// TwinCAT 3 PLC project Untitled1
// ProgramVersion: 3.1.4024.0
// libraries:
//   Tc2_Standard, * (Beckhoff Automation GmbH)
//   Tc2_System, * (Beckhoff Automation GmbH)
//   Tc3_Module, * (Beckhoff Automation GmbH)
// project tree:
//   Actuator/Actuator/ FB_Actuator.TcPOU (not stored)
//   Actuator/DUTs/ E_ActuatorCommand.TcDUT, ST_Inputs.TcDUT, ST_Outputs.TcDUT, ST_ActuatorStatus.TcDUT (not stored), ST_ActuatorConfiguration.TcDUT (not stored)
//   Actuator/GVLs/ Param_Actuator.TcGVL
//   Actuator/ ITF_Actuator.TcIO (not stored)
//   Error/DUTs/ E_ErrorPriority.TcDUT, ST_Error.TcDUT
//   Error/GVLs/ Param_Error.TcGVL
//   Error/POUs/ F_ClearError.TcPOU, F_ResetErrorList.TcPOU
//   / PlcTask.TcTTO
//   POUs/ MAIN.TcPOU (not stored)
// real-time tasks:
//   TASK PlcTask: cycle T#10ms, priority 20, ADS port 350

CONFIGURATION Untitled1
    RESOURCE PLC ON TwinCAT3
        TASK PlcTask(INTERVAL := T#10ms, PRIORITY := 20);
        PROGRAM MAIN WITH PlcTask : MAIN;
    END_RESOURCE
END_CONFIGURATION

// ---- Actuator/DUTs/E_ActuatorCommand.TcDUT
{attribute 'qualified_only'}
{attribute 'strict'}
TYPE E_ActuatorCommand :
(
	Advance := 1,
	Retract := 2
);
END_TYPE

// ---- Actuator/DUTs/ST_Inputs.TcDUT
TYPE ST_Inputs :
STRUCT
	Advanced   AT %I*: BOOL; //Hardware Feedback for Output Advance
	Retracted  AT %I*: BOOL; //Hardware Feedback for Input Retract
END_STRUCT
END_TYPE

// ---- Actuator/DUTs/ST_Outputs.TcDUT
TYPE ST_Outputs :
STRUCT
	Advance   AT %Q*: BOOL; //Hardware Output Advance Signal
	Retract  AT %Q*: BOOL;  //Hardware Output Retract Signal
END_STRUCT
END_TYPE

// ---- Error/DUTs/E_ErrorPriority.TcDUT
{attribute 'qualified_only'}
{attribute 'strict'}
TYPE E_ErrorPriority :
(
	Diagnostic := 0,
	Low := 1,
	Medium := 2,
	High := 3,
	Critical := 4
);
END_TYPE

// ---- Error/DUTs/ST_Error.TcDUT
TYPE ST_Error :
STRUCT
	Active : BOOL := FALSE;
	Label : STRING(Param_Error.LABEL_LEN);
	Message : STRING(Param_Error.MESSAGE_LEN);
	Priority : E_ErrorPriority := E_ErrorPriority.Diagnostic;
END_STRUCT
END_TYPE

// ---- Actuator/GVLs/Param_Actuator.TcGVL
{attribute 'qualified_only'}
VAR_GLOBAL CONSTANT
	DESCRIPTION_LEN : USINT := 40;
	MESSAGE_LEN : UDINT := 255;
	TIMEOUT_LABEL : STRING(Param_Error.LABEL_LEN) := 'Feedback Timeout';
	TIMEOUT_PRIORITY : E_ErrorPriority := E_ErrorPriority.HIGH;
END_VAR

// ---- Error/GVLs/Param_Error.TcGVL
{attribute 'qualified_only'}
VAR_GLOBAL CONSTANT
	LABEL_LEN : USINT := 40;
	MESSAGE_LEN : USINT := 255;
END_VAR

// ---- Error/POUs/F_ClearError.TcPOU
FUNCTION F_ClearError 
VAR_INPUT
	Error : REFERENCE TO ST_Error;
END_VAR
VAR
END_VAR

IF __ISVALIDREF(Error) THEN 
	Error.Active := FALSE;
	Error.Label := '';
	Error.Message := '';
	Error.Priority := E_ErrorPriority.Diagnostic;
END_IF

END_FUNCTION

// ---- Error/POUs/F_ResetErrorList.TcPOU
FUNCTION F_ResetErrorList 
VAR_INPUT
	FirstElement : POINTER TO ST_Error;
	NumElements : UDINT;
END_VAR
VAR
	i : UDINT;
	Instance : POINTER TO ST_Error;
END_VAR

IF FirstElement = 0 THEN 
	RETURN;
END_IF


FOR i := 0 TO (NUMElements - 1) BY 1 DO
	Instance := FirstElement + (i*SIZEOF(firstelement^));
	Instance^.Active := FALSE;
END_FOR

END_FUNCTION
